// TwinCAT 3 PLC project TestSetup
// ProgramVersion: 3.1.4024.0
// libraries:
//   Tc2_Standard, * (Beckhoff Automation GmbH)
//   Tc2_System, * (Beckhoff Automation GmbH)
//   Tc3_Module, * (Beckhoff Automation GmbH)
// project tree:
//   DUTs/ TunePhase.TcDUT
//   / GlobalTextList.TcGTLO, IOTask.TcTTO, PlcTask.TcTTO, Visualization Manager.TcVMO (not stored)
//   GVLs/ GVL.TcGVL
//   POUs/ CheckStability.TcPOU, ConvertIO.TcPOU, MAIN.TcPOU, ParallelPID.TcPOU, Skogestad.TcPOU, TestRealPower.TcPOU
//   VISUs/ Visualization.TcVIS
// real-time tasks:
//   TASK PlcTask: cycle T#10ms, priority 20, ADS port 350
//   TASK IOTask: cycle T#10ms, priority 1, ADS port 351
// I/O:
//   DEVICE Device 5 (EtherCAT), AmsNetId 192.168.18.101.6.1
//     Term 1 (EK1100) [EK1100 EtherCAT Coupler (2A E-Bus)]
//       Term 2 (EL1008) [EL1008 8Ch. Dig. Input 24V, 3ms]
//       Term 3 (EL2008) [EL2008 8Ch. Dig. Output 24V, 0.5A]
//       Term 4 (EL3314) [EL3314 4Ch. Ana. Input Thermocouple (TC)]
//       Term 6 (EL9011) [EL9011 End Terminal]
//     Box 5 (NRGC-ECAT) [NRGC-ECAT]
//       modules: Module 1 (RGC1P60CM32GEN)
// variable links:
//   TestSetup Instance <-> Device 5 (EtherCAT)/Box 5 (NRGC-ECAT)
//     IOTask Inputs/ConvertIO.wRealPower <-> Module 1 (RGC1P60CM32GEN)/TxPDO/Real power reading
//     IOTask Outputs/ConvertIO.byHeaterActuator <-> Module 1 (RGC1P60CM32GEN)/RxPDO/Control level
//   TestSetup Instance <-> Device 5 (EtherCAT)/Term 1 (EK1100)/Term 4 (EL3314)
//     IOTask Inputs/ConvertIO.iTemperatureSensor <-> TC Inputs Channel 1/Value

CONFIGURATION TestSetup
    RESOURCE PLC ON TwinCAT3
        TASK IOTask(INTERVAL := T#10ms, PRIORITY := 1);
        TASK PlcTask(INTERVAL := T#10ms, PRIORITY := 20);
        PROGRAM ConvertIO WITH IOTask : ConvertIO;
        PROGRAM MAIN WITH PlcTask : MAIN;
    END_RESOURCE
END_CONFIGURATION

// ---- DUTs/TunePhase.TcDUT
{attribute 'qualified_only'}
{attribute 'strict'}
TYPE TunePhase :
(
	init,
	baseline,
	step,
	processData,
	done
);
END_TYPE

// ---- GVLs/GVL.TcGVL
{attribute 'qualified_only'}
VAR_GLOBAL PERSISTENT
	// PID variables are stored so the tuner does not have to run each time
	kp: REAL := 0.196;
	ki: REAL := 0.00326;
	kd: REAL := 0;
END_VAR

VAR_GLOBAL
	iHeaterActuator: INT := 0;	// Heater power (0-100%)
	rSetpoint: REAL := 0.0;	// Target temperature (°C)
	
	rTempSensor: REAL := 0.0;	// Temperature (°C)
	iRealPower: INT := 0;		// Actual heater power (W)
	
	doTuning: BOOL := TRUE; 	// Whether or not to run the tuner
END_VAR

// ---- POUs/ConvertIO.TcPOU
PROGRAM ConvertIO
VAR
	wRealPower AT %I*: WORD := 0;
	iTemperatureSensor AT %I*: INT := 0;
	byHeaterActuator AT %Q*: BYTE := 0;
	
	convertedActuator: INT := 0;
END_VAR

GVL.rTempSensor := INT_TO_REAL(iTemperatureSensor) / 10;
GVL.iRealPower := WORD_TO_INT(wRealPower);
byHeaterActuator := REAL_TO_BYTE((GVL.iHeaterActuator * 50) / 100);

END_PROGRAM

// ---- POUs/MAIN.TcPOU
PROGRAM MAIN
VAR
	previousTime: ULINT := 0;
	currentTime: ULINT := 0;
	
	loTime: ULINT := 0;
	hiTime: ULINT := 0;
	getTime: GETSYSTEMTIME;
	
	deltaTime: REAL := 0.0;
	
	skogestadPID: Skogestad( iTest1:=5) ;
	parallelPID: ParallelPID;
	
	init: BOOL := TRUE;
END_VAR

// Get current system time
getTime(timeLoDW => loTime, timeHiDW => hiTime);
currentTime := SHL(hiTime, 32) + loTime;

// Calculate deltaTime
IF previousTime = 0 THEN
    previousTime := currentTime;
	RETURN;
ELSE
    deltaTime := ULINT_TO_REAL(currentTime - previousTime) / 10000000;
    previousTime := currentTime;
END_IF

// Execute skogestad if we should be tuning
IF GVL.doTuning THEN
	skogestadPID(
		rFeedbackVariable := GVL.rTempSensor,
		rSetpoint := GVL.rSetpoint,
		rDeltaTime := deltaTime,
		iOutput => GVL.iHeaterActuator
	);	
ELSE
	parallelPID(
		rFeedbackVariable := GVL.rTempSensor,
		rSetpoint := GVL.rSetpoint,
		rDeltaTime := deltaTime,
		iOutput => GVL.iHeaterActuator
	);
	// TestRealPower(currentOutput => GVl.iHeaterActuator);
END_IF

END_PROGRAM

// ---- POUs/Skogestad.TcPOU
FUNCTION_BLOCK Skogestad EXTENDS ParallelPID
VAR_INPUT
    // Set in superclass
END_VAR
VAR_OUTPUT
    // Set in superclass
END_VAR

VAR
    loadConfig: BOOL := TRUE; 		// Use stored system dynamics if true

    k1: REAL := 3.0;				
    lambda: REAL := 0.0;    		// Measured dead time or delta time
	
	// Stability check
	checkStability: CheckStability;
    rStableWaitTime: REAL := 20;
	runningStableThreshold: REAL := 0.1;
    stabilized: BOOL := FALSE;
    stableTemp: REAL := 0;
    
	// Controller output
	currentOutput: INT := 0;
    baselineOutput: INT := 4;
    stepOutput: INT := 6;
	
	// System dynamics measurement data
    arTemp: ARRAY[0..10000] OF REAL;
    arTime: ARRAY[0..10000] OF REAL;
    currentIndex: INT := 0;
	
    // Variables for asynchronous batch writing
    batchWritePending: BOOL := FALSE;
	batchSize: INT := 10;
    batchTemp: ARRAY[0..10] OF REAL;  // holds one batch of temp data
    batchTime: ARRAY[0..10] OF REAL;  // holds one batch of time data
	validEntries: INT := 0;
	lastTemp: REAL := 0.0;
	skippedTime: REAL := 0.0;
	
	waitTime: REAL := 0.0;

	// Processing variables
    lowestTemp: REAL := 9999;
    baselineTime: REAL := 0;
    measureTemp: REAL := 0;
    initTemp: REAL := 0.0;
	i: INT := 0;
	deadTimeFound: BOOL := FALSE;
	riseStarted: BOOL := FALSE;

    tuningPhase: TunePhase := TunePhase.init; 	// Current tuning phase
END_VAR
VAR PERSISTENT 
    // Store measured system dynamics for recalculation
    riseTime: REAL := 0;
    k: REAL := 0;
    deadTime: REAL := 0;
	
	// Temperature step-response variables
    baselineTemp: REAL := 0.0;
    stepTemp: REAL := 0.0;

END_VAR
// Use temporary arrays for the batch.
VAR_TEMP
	j: INT;
END_VAR

// If a batch write is pending, call M_WriteData repeatedly until it returns TRUE.
IF batchWritePending THEN
    // M_WriteData is asynchronous. It must be called each cycle until it returns TRUE.
    IF M_WriteData(validEntries := validEntries, tempData := batchTemp, timeData := batchTime, clearFile := FALSE) THEN
         batchWritePending := FALSE;
    END_IF;
END_IF;

IF tuningPhase = TunePhase.baseline OR tuningPhase = TunePhase.step THEN
	// Check for stability during baseline and step phases
	checkStability(rCurrentValue := rFeedbackVariable, 
				   rDeltaTime := rDeltaTime, 
				   rThreshold := runningStableThreshold, 
				   rDuration := 30,
				   rInitialValue := -99.9, 
				   bIsStable => stabilized);
	
	// Save data in batches during baseline and step phases			   
	IF NOT (lastTemp = rFeedbackVariable)
		AND NOT batchWritePending THEN
		lastTemp := rFeedbackVariable;
		batchTemp[currentIndex] := rFeedbackVariable;
		batchTime[currentIndex] := INT_TO_REAL(REAL_TO_INT(skippedTime * 100.0 + 0.05)) / 100.0;
		skippedTime := 0;
		validEntries := currentIndex;
		
		currentIndex := currentIndex + 1;
		IF currentIndex > batchSize THEN
			batchWritePending := TRUE;
			currentIndex := 0;
		END_IF
	ELSE
		skippedTime := skippedTime + rDeltaTime;
	END_IF
	
END_IF

CASE tuningPhase OF
TunePhase.init:

	currentOutput := 0; // Ensure output is off
	
	IF loadConfig THEN
		tuningPhase := TunePhase.processData;	// Skip tuning if using stored variables
		RETURN;
	END_IF
	
    // Wait for stabilization before starting tuning.
    checkStability(rCurrentValue := rFeedbackVariable, 
                   rDeltaTime := rDeltaTime, 
                   rThreshold := 0.2, 
                   rDuration := 30,
                   rInitialValue := -99.9, 
                   bIsStable => stabilized);
    IF stabilized THEN
		M_WriteData(validEntries := validEntries, tempData := batchTemp, timeData := batchTime, clearFile := TRUE); // Clear data file
        tuningPhase := TunePhase.baseline;
		currentOutput := baselineOutput;
		initTemp := rFeedbackVariable;
		lastTemp := rFeedbackVariable;
        stabilized := FALSE;
    ELSE
        RETURN;
    END_IF

TunePhase.baseline:

	IF stabilized THEN
		tuningPhase := TunePhase.step;
        currentOutput := stepOutput;
		baselineTemp := rFeedbackVariable;
		initTemp := rFeedbackVariable;
        stabilized := FALSE;
    END_IF
	
TunePhase.step:

	IF stabilized THEN
		IF NOT (currentIndex = 0) THEN
			batchWritePending := TRUE;
			validEntries := currentIndex;
		END_IF;	
	
        stepTemp := rFeedbackVariable;
		currentOutput := 0;
		tuningPhase := TunePhase.processData;
    END_IF
	
TunePhase.processData:

	// Wait for the batch to finish writing before processing data
	IF batchWritePending THEN
		RETURN;
	END_IF
	
	validEntries := 0;
	
    IF M_ReadData(tempData => batchTemp, timeData => batchTime, validEntries => validEntries) THEN
		IF NOT (validEntries = 0) THEN 
			
			FOR i := 0 TO validEntries - 1 DO
				IF NOT deadTimeFound THEN
					IF batchTemp[i] < lowestTemp THEN
						lowestTemp := batchTemp[i];
					END_IF;
					IF batchTemp[i] > lowestTemp + 0.002 * (stepTemp - lowestTemp) THEN
						deadTimeFound := TRUE;
					ELSE
						deadTime := deadTime + batchTime[i];
					END_IF;
				END_IF;
	
				riseTime := riseTime + batchTime[i];
				IF NOT riseStarted AND batchTemp[i] > baselineTemp THEN 
					baselineTime := riseTime;
					riseStarted := TRUE;
				END_IF;
				
				IF batchTemp[i] > baselineTemp + 0.632 * (stepTemp - baselineTemp) THEN
					riseTime := riseTime - baselineTime;
					tuningPhase := TunePhase.done;
					EXIT;
				END_IF;
			END_FOR;
			
		END_IF;		

    END_IF;

TunePhase.done:

	// Calculate final PID gains.
    k1 := riseTime / (deadTime + deadTime);
    lambda := MAX(deadTime, rDeltaTime);
    GVL.kp := riseTime / (k * (lambda + deadTime));
    GVL.ki := GVL.kp / MIN(riseTime, k1 * (lambda + deadTime));
    GVL.kd := 0;
	
	GVL.doTuning := FALSE; // Let PID controller take over
	
END_CASE

iOutput := currentOutput;

METHOD PRIVATE M_ReadData : BOOL
VAR_OUTPUT
    tempData : ARRAY[0..10] OF REAL;
    timeData : ARRAY[0..10] OF REAL;
    validEntries : INT;
END_VAR
VAR
    sPath   : STRING(80) := 'C:\Temp\DataLog.txt';
    sNetId  : T_AmsNetId := ''; // Target system (empty is local)
    
    hashPos : INT;
    tempStr : STRING(100);
    timeStr : STRING(100);
    tempVals: ARRAY[0..10] OF STRING(10);
    timeVals: ARRAY[0..10] OF STRING(10);
    i       : INT;
END_VAR

VAR_STAT
	hFile   : UINT;
    sLine   : STRING(255);	

	fbOpen  : FB_FileOpen;
    fbRead  : FB_FileGets;
    fbClose : FB_FileClose;	

	state   : INT := 0;  // 0: open, 1: read, 2: close, 3: done/error
	
	waitCounter : INT := 0;
	returnState: INT := 0;
END_VAR
CASE state OF
0:  // Open file (needs to run 1 cycle)
    fbOpen(bExecute:=FALSE);
	fbOpen(sNetId:=sNetId, sPathName:=sPath, nMode:=FOPEN_MODEREAD, ePath:=PATH_GENERIC, bExecute:=TRUE);
    state := 1;
	returnState := 1;
	
1:	// Open file (after 1 cycle)
	fbOpen(bExecute:=FALSE);
	IF NOT fbOpen.bBusy THEN
        IF fbOpen.bError THEN
            state := 5;
            M_ReadData := FALSE;
        ELSE
            hFile := fbOpen.hFile;
            state := 2;
        END_IF;
        fbOpen(bExecute:=FALSE);
    END_IF;
	
2:	// Read line (needs 1 cycle)
	fbRead(sNetId:=sNetId, hFile:=hFile, sLine=>sLine, bExecute:=FALSE);
	state := 100; // Wait phase
	returnState := 3;

3:  // Read line (after 1 cycle)
    fbRead(sNetId:=sNetId, hFile:=hFile, sLine=>sLine, bExecute:=TRUE);
    IF NOT fbRead.bBusy THEN
        IF fbRead.bError OR fbRead.bEOF THEN
            state := 4; // Done or error
        ELSE
			IF sLine = '' THEN
				state := 2;
				M_ReadData := FALSE;
				RETURN;
			END_IF
            hashPos := FIND(sLine, '#'); // # is the seperator between temp and time data
            tempStr := LEFT(sLine, hashPos - 1); // Temperature data
            timeStr := RIGHT(sLine, LEN(sLine) - hashPos); // Time data

            validEntries := SplitCSV(tempStr, ADR(tempVals));
            FOR i := 0 TO validEntries - 1 DO
                tempData[i] := STRING_TO_REAL(tempVals[i]);
            END_FOR

            validEntries := SplitCSV(timeStr, ADR(timeVals));
            FOR i := 0 TO validEntries - 1 DO
                timeData[i] := STRING_TO_REAL(timeVals[i]);
            END_FOR

			state := 2;
            M_ReadData := TRUE;
            RETURN; // New batch processed, return true each batch
        END_IF;
        fbRead(bExecute:=FALSE);
    END_IF;

4:  // Close file
    fbClose(sNetId:=sNetId, hFile:=hFile, bExecute:=TRUE);
    IF NOT fbClose.bBusy THEN
        fbClose(bExecute:=FALSE);
        state := 5;
    END_IF;

5:  // Done/Error
    M_ReadData := FALSE;
	
100: // Wait
	IF waitCounter < 10 THEN
		waitCounter := waitCounter + 1;
	ELSE
		waitCounter := 0;
		state := returnState;
	END_IF

END_CASE;
END_METHOD

METHOD PRIVATE M_WriteData : BOOL
VAR_INPUT
	validEntries: INT := 0;
    tempData: ARRAY[0..10] OF REAL;
    timeData: ARRAY[0..10] OF REAL;
	clearFile: BOOL := FALSE;
END_VAR
VAR
    sPath   : STRING(80) := 'C:\Temp\DataLog.txt';
    sNetId  : T_AmsNetId := '';  // Target system (empty is local)
    i       : INT;
END_VAR
VAR_STAT
	sLine   : STRING(255);
	hFile   : UINT;
	fbOpen : FB_FileOpen;
    fbWrite: FB_FileWrite;
    fbClose: FB_FileClose;
    state : INT := 0;  // 0: open, 1: write temp, 2: write time, 3: close, 4: error
END_VAR
CASE state OF
    0: 
		IF NOT clearFile THEN
			 // Open file in append mode
			 fbOpen(
				 sNetId := sNetId,
				 sPathName := sPath,
				 nMode := FOPEN_MODEAPPEND OR FOPEN_MODETEXT,
				 ePath := PATH_GENERIC,
				 bExecute := TRUE
			 );
			 IF NOT fbOpen.bBusy THEN
				 IF fbOpen.bError THEN
					 state := 4;
					 M_WriteData := FALSE;
				 ELSE
					 hFile := fbOpen.hFile;
					 state := 1;
				 END_IF;
				 fbOpen(bExecute := FALSE);
			 END_IF;
		ELSE
			// Clears the contents of the file
			fbOpen(
				 sNetId := sNetId,
				 sPathName := sPath,
				 nMode := FOPEN_MODEWRITE OR FOPEN_MODETEXT,
				 ePath := PATH_GENERIC,
				 bExecute := TRUE
			 );
			 IF NOT fbOpen.bBusy THEN
				 IF fbOpen.bError THEN
					 state := 4;
					 M_WriteData := FALSE;
				 ELSE
					 hFile := fbOpen.hFile;
					 state := 3; // Only clear contents
				 END_IF;
				 fbOpen(bExecute := FALSE);
			 END_IF;
		END_IF

         
    1: // Build CSV line: tempData values, '#' delimiter, then timeData values, then newline
		// Each new line represents a batch
         sLine := '';
         // Append tempData values
         FOR i := 0 TO validEntries - 1 DO
             sLine := CONCAT(sLine, REAL_TO_STRING(tempData[i]));
             IF i < validEntries - 1 THEN
                 sLine := CONCAT(sLine, ',');
             END_IF;
         END_FOR;
		 
         // Append delimiter
         sLine := CONCAT(sLine, '#');
         
         fbWrite(
             sNetId := sNetId,
             hFile := hFile,
             pWriteBuff := ADR(sLine),
             cbWriteLen := INT_TO_UDINT(LEN(sLine)),
             bExecute := TRUE
         );
         IF NOT fbWrite.bBusy THEN
             IF fbWrite.bError THEN
                 state := 4;
                 M_WriteData := FALSE;
             ELSE
                 state := 2;
             END_IF;
             fbWrite(bExecute := FALSE);
         END_IF;
    2:
		sLine := ''; // Clear string
			
		// Append timeData values
		FOR i := 0 TO validEntries - 1 DO
		 sLine := CONCAT(sLine, REAL_TO_STRING(timeData[i]));
		 IF i < validEntries - 1 THEN
			 sLine := CONCAT(sLine, ',');
		 END_IF;
		END_FOR;
		
		// Append newline
		sLine := CONCAT(sLine, '$n');
		
		// Write line (batch) to file
		fbWrite(
             sNetId := sNetId,
             hFile := hFile,
             pWriteBuff := ADR(sLine),
             cbWriteLen := INT_TO_UDINT(LEN(sLine)),
             bExecute := TRUE
         );
         IF NOT fbWrite.bBusy THEN
             IF fbWrite.bError THEN
                 state := 4;
                 M_WriteData := FALSE;
             ELSE
                 state := 3;
             END_IF;
             fbWrite(bExecute := FALSE);
         END_IF;
    3: // Close file
         fbClose(
             sNetId := sNetId,
             hFile := hFile,
             bExecute := TRUE
         );
         IF NOT fbClose.bBusy THEN
             fbClose(bExecute := FALSE);
             state := 0;
             M_WriteData := TRUE;
         END_IF;
         
    4: // Error: reset state
         state := 0;
         M_WriteData := FALSE;
END_CASE;
END_METHOD

METHOD PRIVATE SplitCSV : INT
VAR_INPUT
    input : STRING(100);
    output: POINTER TO ARRAY[0..10] OF STRING(10);
END_VAR
VAR
    i, count, commaPos: INT;
    remaining: STRING(100);
END_VAR
remaining := input;
count := 0;

WHILE LEN(remaining) > 0 AND count < 10 DO
    commaPos := FIND(remaining, ',');
    IF commaPos = 0 THEN
        output^[count] := remaining;
        remaining := '';
    ELSE
        output^[count] := LEFT(remaining, commaPos - 1);
        remaining := RIGHT(remaining, LEN(remaining) - commaPos);
    END_IF
    count := count + 1;
END_WHILE

SplitCSV := count;
END_METHOD

END_FUNCTION_BLOCK

// ---- POUs/ParallelPID.TcPOU
FUNCTION_BLOCK ParallelPID
VAR_INPUT
	rFeedbackVariable: REAL := 0.0; // The measured temperature (°C)
	rSetpoint: REAL := 0.0; 		// The target temperature (°C)
	rDeltaTime: REAL := 0.0;		// The cycle's run time (S)
END_VAR
VAR_OUTPUT
	iOutput: INT := 0; 				// The controller output (0% - 100%)
END_VAR
VAR
	MAX_OUTPUT: INT := 100;			// Highest possible controller output (%)
	MIN_OUTPUT: INT := 0;			// Lowest possible controller output (%)
	
	lastOutput: INT := 0;
	
	error: REAL := 0.0;				// Current error
	prevError: REAL := 0.0;			// Last calculated error
	
	integral: REAL := 0.0;			// Previous iteration's integral
	rollbackIntegral: REAL := 0.0;	// This iterations integral for rollback
END_VAR

error := rSetpoint - rFeedbackVariable;
rollbackIntegral := integral;
integral := integral + error * rDeltaTime;

iOutput := REAL_TO_INT(GVL.kp * error
						+ GVL.ki * integral
						+ GVL.kd * (error - prevError) / rDeltaTime);

prevError := error;

IF iOutput >= MAX_OUTPUT THEN
	iOutput := MAX_OUTPUT;
	integral := rollbackIntegral;
ELSIF iOutput <= MIN_OUTPUT THEN
	iOutput := MIN_OUTPUT;
	integral := rollbackIntegral;
END_IF
				
lastOutput := iOutput;

END_FUNCTION_BLOCK

// ---- POUs/CheckStability.TcPOU
FUNCTION_BLOCK CheckStability
VAR_INPUT
    rCurrentValue : REAL;     // New measurement to add
    rDeltaTime    : REAL;     // Cycle time (dt) in seconds
    rThreshold    : REAL;     // Allowed range for stability
    rDuration     : REAL;     // Desired stability duration, max 60 (seconds)
    rInitialValue : REAL;     // Initial value (to detect resets)
END_VAR
VAR_OUTPUT
    bIsStable         : BOOL;   // TRUE if the buffer is stable
END_VAR
VAR
    stable_samples_required : INT;
    i                       : INT;
    rMax                    : REAL;
    rMin                    : REAL;
    sum                     : REAL;
    num_to_average          : INT;
    lastInitial             : REAL := -99.9; // remembers previous initial value
    currentIndex            : INT := 0;     // current count of samples in buffer
    stableBuffer            : ARRAY[0..6000] OF REAL; // fixed‐size buffer (simulate FIFO)
    emptyBuffer             : ARRAY[0..6000] OF REAL; // for resetting the buffer
	rStableCounter : REAL := 0.0; // Accumulated stable time
	
	init: BOOL := TRUE;
END_VAR

IF init THEN
	init := FALSE;
	// Calculate how many samples are needed to span the desired duration.
	stable_samples_required := REAL_TO_INT(rDuration / rDeltaTime);
END_IF

// When overall stability is achieved, reset the buffer AND counter:
IF bIsStable THEN
     stableBuffer := emptyBuffer;
     currentIndex := 0;
     rStableCounter := 0.0;
END_IF

// If the initial value has changed, reset the buffer.
IF rInitialValue <> lastInitial THEN
    lastInitial := rInitialValue;
    currentIndex := 0;
    stableBuffer := emptyBuffer;
	rStableCounter := 0;
END_IF

IF ABS(rInitialValue - rCurrentValue) < 1.0 THEN
    // If deviation is too low, reset the buffer.
    currentIndex := 0;
    stableBuffer := emptyBuffer;
	rStableCounter := 0;
END_IF

// Append new value using FIFO logic:
IF currentIndex < stable_samples_required THEN
    stableBuffer[currentIndex] := rCurrentValue;
    currentIndex := currentIndex + 1;
ELSE
    // Shift buffer left by one element.
    FOR i := 0 TO stable_samples_required - 2 DO
        stableBuffer[i] := stableBuffer[i + 1];
    END_FOR
    stableBuffer[stable_samples_required - 1] := rCurrentValue;
END_IF

// Only check stability if the buffer is full.
IF currentIndex = stable_samples_required THEN
    rMax := stableBuffer[0];
    rMin := stableBuffer[0];
    FOR i := 1 TO stable_samples_required - 1 DO
        IF stableBuffer[i] > rMax THEN
            rMax := stableBuffer[i];
        END_IF
        IF stableBuffer[i] < rMin THEN
            rMin := stableBuffer[i];
        END_IF
    END_FOR
    bIsStable := ((rMax - rMin) < rThreshold + 0.01);
ELSE
    bIsStable := FALSE;
END_IF

// Now update the timer:
IF bIsStable THEN
    rStableCounter := rStableCounter + rDeltaTime;
ELSE
    rStableCounter := 0.0;
END_IF

// Only keep overall stability true if stable condition has been met for at least half of rDuration:
IF rStableCounter >= (rDuration / 2.0) THEN
    bIsStable := TRUE;
ELSE
    bIsStable := FALSE;
END_IF

END_FUNCTION_BLOCK

// ---- POUs/TestRealPower.TcPOU
PROGRAM TestRealPower
VAR
	currentCycle: INT := 0;
	cycleCount: INT := 0;
	switch: BOOL := FALSE;
	
END_VAR
VAR_OUTPUT
	currentOutput: INT := 0;
END_VAR

IF currentCycle < GVL.cyclesToSkip THEN
	currentCycle := currentCycle + 1;
	RETURN; // Skip cycle
ELSE
	currentCycle := 0;
END_IF

cycleCount := cycleCount + 1;

IF NOT switch AND currentOutput = 100 THEN
	switch := TRUE;
END_IF

IF cycleCount >= 25 THEN
	IF switch THEN
		currentOutput := currentOutput - 10;
	ELSE
		currentOutput := currentOutput + 10;
	END_IF
	
	cycleCount := 0;
END_IF

END_PROGRAM

// ---- GlobalTextList.TcGTLO
TEXTLIST GlobalTextList
  70 = ''
  326 = '                                                                                                                                                                                                                                                                                   %'
  575 = '                                                                                                                                                                                                                                                                               %'
  22 = '                                                                                                                                                                                                                             %'
  783 = '                                                                                                          %'
  333 = '  °C'
  161 = '%'
  395 = 'Controller output (%)'
  259 = 'Controller output%'
  724 = 'Real Power Reading (W)'
  384 = 'Setpoint        (°C)'
  478 = 'Setpoint       (°C)'
  432 = 'Setpoint      (°C)'
  703 = 'Setpoint (°C)'
  252 = 'Skogestad Tuner on Test Setup'
  823 = 'Skogestad Tunerr on Test Setup'
  382 = 'Temperature (°C)'
  609 = '\\n %'
  957 = '°C'
END_TEXTLIST

// ---- VISUs/Visualization.TcVIS
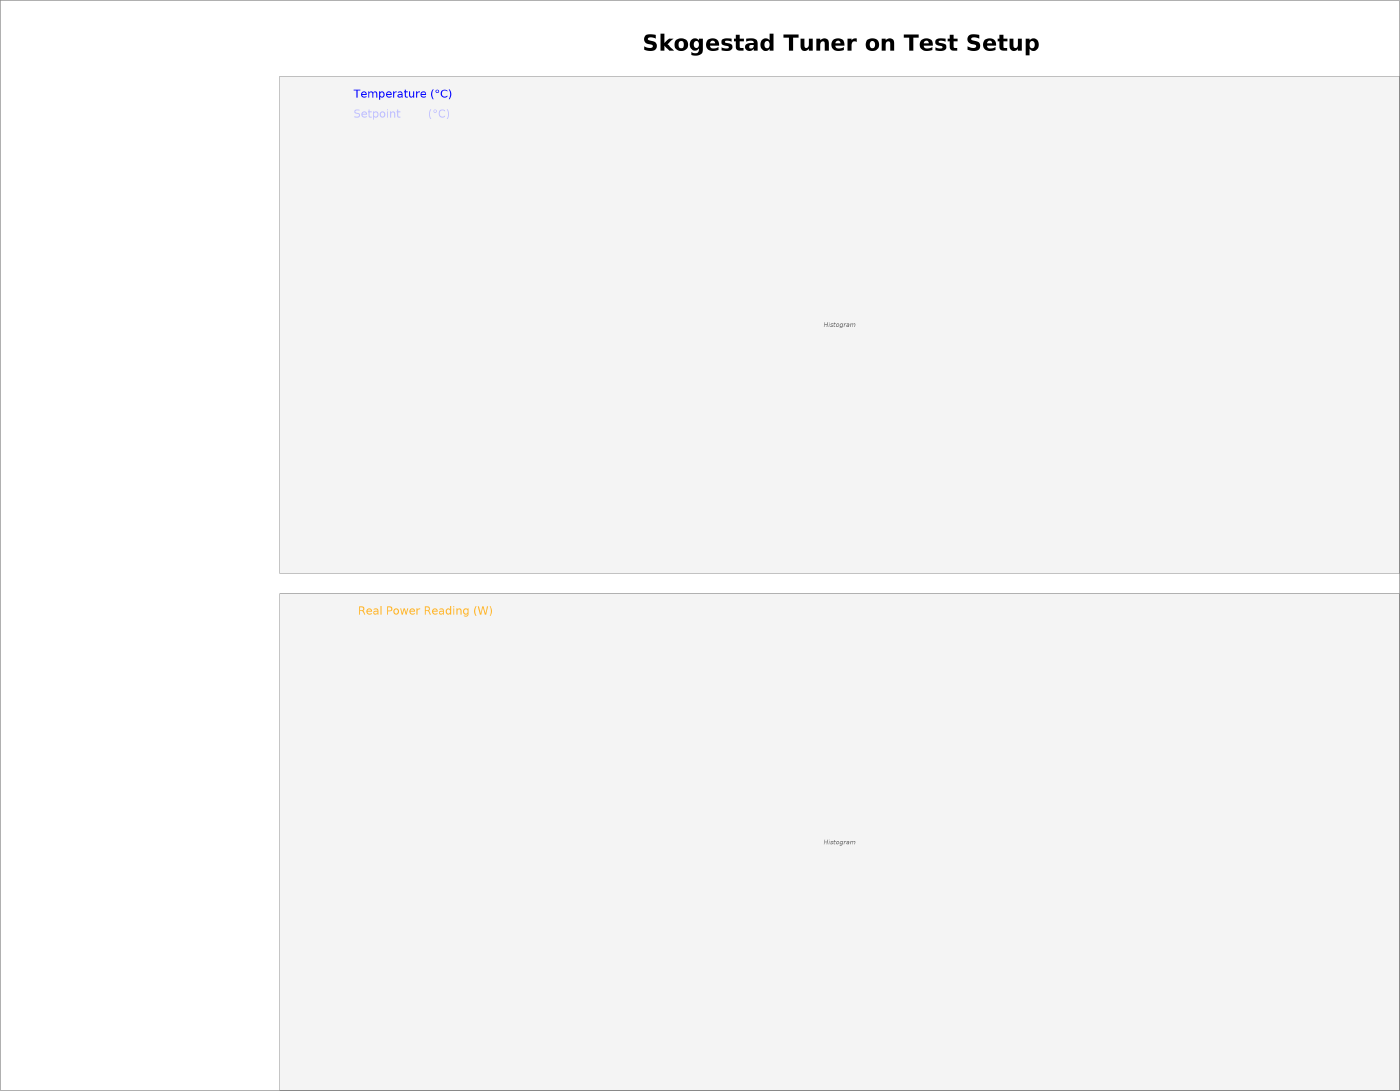
VISUALIZATION Visualization  // 2249x1754
    Histogram (449,122 1800x800), scale format: %.1f, scale 0..100
        p1518820177: GVL.arSetpointData
        p102497268: GVL.arSetpointData
        p788070771: ARRAY [0..20000] OF REAL
    Histogram (449,122 1800x800), scale format: %.1f, scale 0..100
        p1518820177: GVL.arTempData
        p102497268: GVL.arTempData
        p788070771: ARRAY [0..2000] OF REAL
    Histogram (449,954 1800x800), scale format: %.1f, scale 0..100
        p1518820177: GVL.arControllerData
        p102497268: GVL.arControllerData
        p788070771: ARRAY [0..2000] OF INT
    Label (565,136 167x30), "Temperature (°C)"
    Label (570,1007 193x30), "Controller output (%)"
    Label (1022,36 659x66), "Skogestad Tuner on Test Setup"
    Histogram (449,954 1800x800), scale format: %.1f, scale 0..100
        p1518820177: GVL.arRealPowerData
        p102497268: GVL.arRealPowerData
        p788070771: ARRAY [0..10000] OF INT
    Label (563,967 232x30), "Real Power Reading (W)"
    Label (565,168 167x30), "Setpoint (°C)"
END_VISUALIZATION
